Fanuc KAREL source: compact_preamble.KL

PROGRAM KT00410
%NOLOCKGROUP
VAR
S1 : STRING[80];S2 : STRING[80];OUT:BOOLEAN
BEGIN
S1='A'
S2='B'
S1='A'
S2='B'
OUT=(S1 > S2)
END KT00410
